// TIA Portal V20 export
// export: Created 2025-12-01T14:56:13.8156468Z, ExportSetting None, DisplayName Totally Integrated Automation Portal, DisplayVersion V20 Update 3, DisplayName TIA Portal Openness, DisplayVersion V20 Update 3, DisplayName TIA Portal Version Control Interface, DisplayVersion V20 Update 3, DisplayName STEP 7 Professional, DisplayVersion V20 Update 3, DisplayName STEP 7 Safety, DisplayVersion V20 Update 2, DisplayName WinCC Basic/Comfort/Advanced, DisplayVersion V20 Update 3, DisplayName WinCC Professional, DisplayVersion V20 Update 3, DisplayName WinCC Unified, DisplayVersion V20 Update 3
TYPE "UDT_EmisionDeDispositivo"
   STRUCT
      Error : UDInt;
      Auxliar_01 : UInt;
      Auxliar_02 : UInt;
      Protocolo { S7_SetPoint := 'True'} : "UDT_ProtocoloEmiDispositivo";
   END_STRUCT;
END_TYPE
